// TIA Portal V19 export
TYPE "LAF_typeAxisMannualParameters"
// stored: Access Published
   STRUCT
      upperVel : LReal := 500.0;   // 手动速度上限
      vel : LReal := 100.0;   // 手动速度设定值，画面做限制根据上限值如果超了不允许输入
      acc : LReal := 1.0;
      dec : LReal := 1.0;
   END_STRUCT;
END_TYPE
